FUNCTION_BLOCK PUBLIC ButtonPress EXTENDS ButtonHMI
VAR_INPUT
END_VAR
VAR_OUTPUT
    outPress       : BOOL;
    outRisingEdge  : BOOL;
    outFallingEdge : BOOL;
END_VAR
VAR
    _clk : BOOL; // used to generate the R_Trig and F_Trig
END_VAR

_disable := inDisable;
_on      := inOn AND NOT inError;
_error   := inError;

outPress       := _button AND NOT inDisable;
outRisingEdge  := _button AND NOT _clk AND NOT inDisable;
outFallingEdge := NOT _button AND _clk AND NOT inDisable;

_clk := _button;

END_FUNCTION_BLOCK

(* stored: Version 1.1.0.1, ProductVersion 3.1.4024.12
   POU ButtonPress: Id {d2dcafbd-5508-4cb2-8df9-57a88efd2ac5}, SpecialFunc None *)
